Omron CX-Programmer project NewProject (CX-Programmer 9.31)

# PLC NewPLC1: CP1L L

## Global symbols (name address type ; comment)
0.00 BOOL  ; On/Off
0.01 BOOL  ; Type A
0.02 BOOL  ; Type B
0.03 BOOL  ; Type C
0.04 BOOL  ; Sensor 1
0.05 BOOL  ; Sensor 2
0.06 BOOL  ; Sensor 3
0.07 BOOL  ; Sensor 4
100.00 BOOL  ; Motor On
100.01 BOOL  ; Solenoid valve 1
100.02 BOOL  ; Solenoid valve 2
100.03 BOOL  ; Solenoid valve 3
100.04 BOOL  ; Trig Barcode
100.05 BOOL  ; Lamp
T0000 BOOL  ; Stand BY
T0001 BOOL  ; Stop conveyor
T0005 BOOL  ; Lamp OFF
T0006 BOOL  ; Lamp ON

## Program NewProgram1 (cyclic task 0)
; Automatic Sorting Production Line Model

### Section Section1

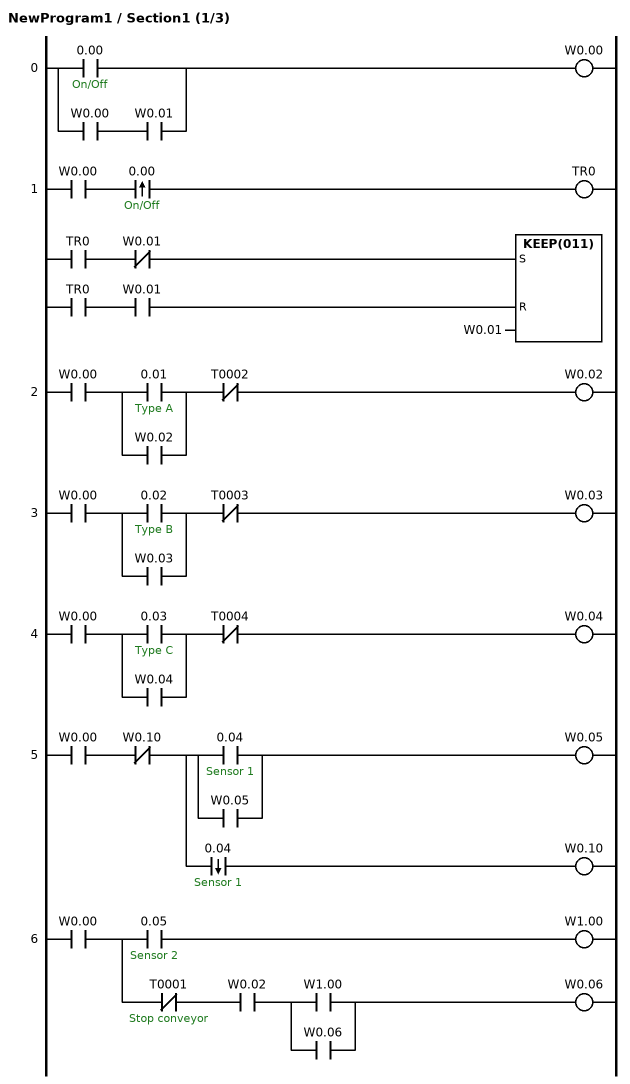
; rung 0
LD 0.00  ; On/Off
LD W0.00
AND W0.01
ORLD
OUT W0.00
; rung 1
LD W0.00
@AND 0.00  ; On/Off
OUT TR0
ANDNOT W0.01
LD TR0
AND W0.01
KEEP(011) W0.01
; rung 2
LD W0.00
LD 0.01  ; Type A
OR W0.02
ANDLD
ANDNOT T0002
OUT W0.02
; rung 3
LD W0.00
LD 0.02  ; Type B
OR W0.03
ANDLD
ANDNOT T0003
OUT W0.03
; rung 4
LD W0.00
LD 0.03  ; Type C
OR W0.04
ANDLD
ANDNOT T0004
OUT W0.04
; rung 5
LD W0.00
ANDNOT W0.10
OUT TR0
LD 0.04  ; Sensor 1
OR W0.05
ANDLD
OUT W0.05
LD TR0
%AND 0.04  ; Sensor 1
OUT W0.10
; rung 6
LD W0.00
OUT TR0
AND 0.05  ; Sensor 2
OUT W1.00
LD TR0
ANDNOT T0001  ; Stop conveyor
AND W0.02
LD W1.00
OR W0.06
ANDLD
OUT W0.06

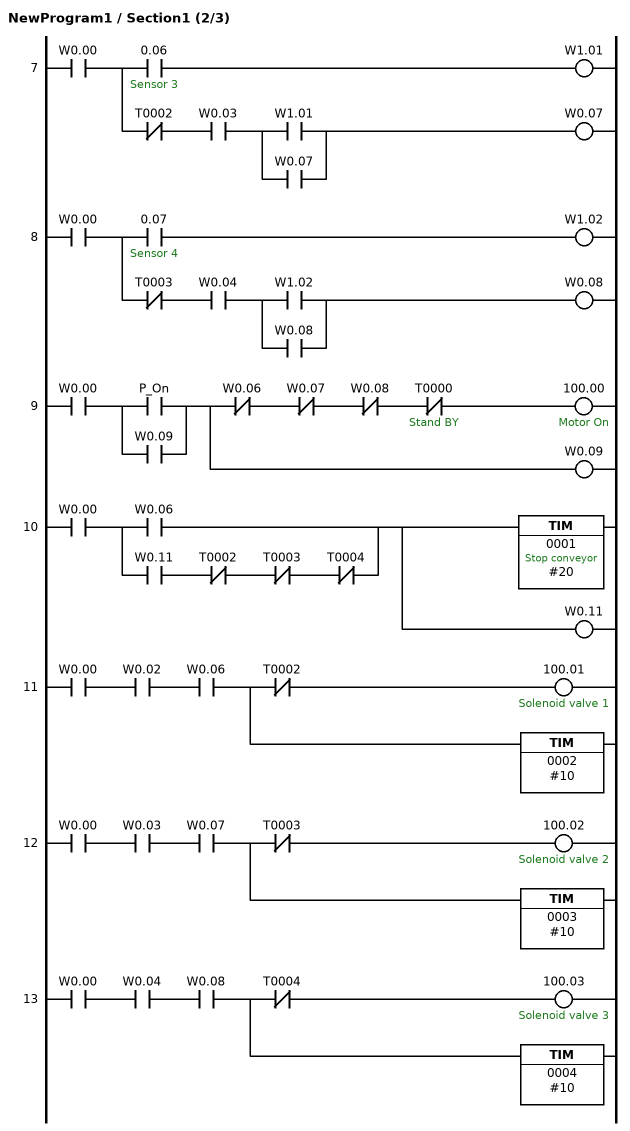
; rung 7
LD W0.00
OUT TR0
AND 0.06  ; Sensor 3
OUT W1.01
LD TR0
ANDNOT T0002
AND W0.03
LD W1.01
OR W0.07
ANDLD
OUT W0.07
; rung 8
LD W0.00
OUT TR0
AND 0.07  ; Sensor 4
OUT W1.02
LD TR0
ANDNOT T0003
AND W0.04
LD W1.02
OR W0.08
ANDLD
OUT W0.08
; rung 9
LD W0.00
LD P_On
OR W0.09
ANDLD
OUT TR0
ANDNOT W0.06
ANDNOT W0.07
ANDNOT W0.08
ANDNOT T0000  ; Stand BY
OUT 100.00  ; Motor On
LD TR0
OUT W0.09
; rung 10
LD W0.00
LD W0.06
LD W0.11
ANDNOT T0002
ANDNOT T0003
ANDNOT T0004
ORLD
ANDLD
TIM 0001 #20  ; Stop conveyor
OUT W0.11
; rung 11
LD W0.00
AND W0.02
AND W0.06
OUT TR0
ANDNOT T0002
OUT 100.01  ; Solenoid valve 1
LD TR0
TIM 0002 #10
; rung 12
LD W0.00
AND W0.03
AND W0.07
OUT TR0
ANDNOT T0003
OUT 100.02  ; Solenoid valve 2
LD TR0
TIM 0003 #10
; rung 13
LD W0.00
AND W0.04
AND W0.08
OUT TR0
ANDNOT T0004
OUT 100.03  ; Solenoid valve 3
LD TR0
TIM 0004 #10

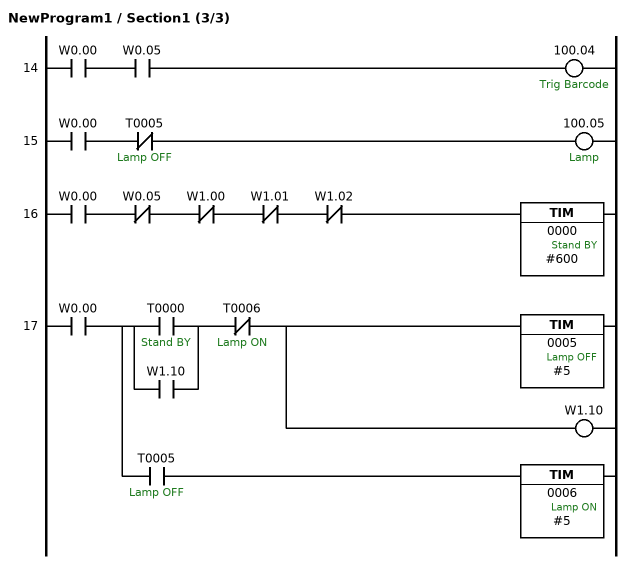
; rung 14
LD W0.00
AND W0.05
OUT 100.04  ; Trig Barcode
; rung 15
LD W0.00
ANDNOT T0005  ; Lamp OFF
OUT 100.05  ; Lamp
; rung 16
LD W0.00
ANDNOT W0.05
ANDNOT W1.00
ANDNOT W1.01
ANDNOT W1.02
TIM 0000 #600  ; Stand BY
; rung 17
LD W0.00
OUT TR0
LD T0000  ; Stand BY
OR W1.10
ANDLD
ANDNOT T0006  ; Lamp ON
TIM 0005 #5  ; Lamp OFF
OUT W1.10
LD TR0
AND T0005  ; Lamp OFF
TIM 0006 #5  ; Lamp ON
; rung 18
END(001)

### Section END
; rung 0
END(001)